FUNCTION_BLOCK FB_NotEnabled
VAR_INPUT
END_VAR
VAR_OUTPUT
END_VAR
VAR
END_VAR

	HMIoutput.bHMIGreenLED := FALSE;
	HMIoutput.bHMIRedLED := FALSE;	
	
	HMIinput.bHMIStartSwitch := FALSE;
	HMIinput.bHMIStopSwitch := FALSE;

END_FUNCTION_BLOCK

(* stored: Version 1.1.0.1, ProductVersion 3.1.4024.10
   POU FB_NotEnabled: Id {e8d87ba8-6bd7-4439-a9f9-582b97ad65c0}, SpecialFunc None *)
